(* IEC 61131-3 sources: CodesysTest/export/UN00 - Sharp Bagger/FB_PackMLStates.pou/ClearingDone.prop, 1 file *)

(* ---- Get.pm.st ---- *)
(*#-#-#-#-#-#-#-#-#-#---Declaration---#-#-#-#-#-#-#-#-#-#-#-#-#*)

VAR
END_VAR
(*#-#-#-#-#-#-#-#-#-#---Implementation---#-#-#-#-#-#-#-#-#-#-#-#-#*)

ClearingDone := _clearingDone;
